(* Logix 5000 project; controller RSL5k_18_Template_noLib Emulate 5570 rev 32.11; software revision 32.02; part 10 of 16 *)
(* tags used below, declared in another part *)
   Inp_UseCVInitVal : ALIAS FOR Wrk_PIDE.CVInitReq;   // 1=Initialize CV to Inp_CVInitValue
   Inp_PVSrcQ : DINT;   // Source and Quality of Inp_PV (enum)
   Inp_PVNotify : DINT;   // PV Alarm Level and Acknowledgement (enum)
   Inp_CVNotify : DINT;   // CV Alarm Level and Acknowledgement (enum)
   Inp_CascSPNotify : DINT;   // Cascade SP Alarm Level and Acknowledgement (enum)
   Inp_IntlkOK : BOOL;   // 1=Interlocks OK, CV can be set
   Inp_NBIntlkOK : BOOL;   // 1=Non-Bypassable Interlocks OK, CV can be set
   Inp_IntlkAvail : BOOL;   // 1 = Interlock Availibility OK
   Cfg_HasRatio : ALIAS FOR Wrk_PIDE.UseRatio;   // 1=Casc Loop Mode is Ratio, 0=Casc Loop Mode is Cascade
   Cfg_InitToMan : ALIAS FOR Wrk_PIDE.ManualAfterInit;   // 1=Go to Manual Loop Mode when an init request is seen
   Cfg_HiHiDevLim : REAL;   // Current High-High Deviation Status Threshold (PVEU)
   Cfg_HiHiDevDB : REAL;   // High-High Devation Status Deadband (PVEU)
   Cfg_HiDevLim : REAL;   // Current High Deviation Status Threshold (PVEU)
   Cfg_HiDevDB : REAL;   // High Devation Status Deadband (PVEU)
   Cfg_LoDevLim : REAL;   // Current Low Deviation Status Threshold (PVEU)
   Cfg_LoDevDB : REAL;   // Low Devation Status Deadband (PVEU)
   Cfg_LoLoDevLim : REAL;   // Current Low-Low Deviation Status Threshold (PVEU)
   Cfg_LoLoDevDB : REAL;   // Low-Low Devation Status Deadband (PVEU)
   Val_PV : REAL;   // Value of Loop PV (PVEU)
   Val_SP : ALIAS FOR Wrk_PIDE.SP;   // Value of SP being used (after ramping and clamping (PVEU)
   SrcQ_IO : DINT;   // Source and Quality of primary I/O (enumeration)
   SrcQ : DINT;   // Source and Quality of primary Val/Sts (enumeration)
   Val_Sts : DINT;   // Loop Status enum: 0=unknown (POoS @ Intlk CV), 1=Manual, 2=Auto, 3=Cascade (no ratio), 4=Ratio
   Val_Fault : DINT;   // Loop Fault: 0=none, 1=PV Uncertain, 22=LoDev, 23=HiDev, 27=LLDev, 28=HHDev, 29=Intlk Trip, 30=SP Fail, 31=PV Fail, 32=CV
   Val_State : DINT;   // Loop State: 0=Man, 1=In DB, 2=Not in DB, 3=SPRamp, 4=CVRamp, 5=Ratio Clamp, 6=SP Clamp, 7=CV Clamp, 8=Windup L, 9=Windup
   Val_NotifyAll : DINT;   // Highest Alarm prio and ack status this object + PV, CV, CascSP (enum)
   Val_UnackAlmC : DINT;   // Count of Unacknowledged Alarms
   Sts_Casc : BOOL;   // 1=Loop Mode is Cascade/Ratio
   Sts_Auto : BOOL;   // 1=Loop Mode is Auto
   Sts_Man : BOOL;   // 1=Loop Mode is Manual
   Sts_Initializing : ALIAS FOR Wrk_PIDE.CVInitializing;   // 1=CV is initializing because of Request from this loop's Secondary
   Sts_WindupHi : ALIAS FOR Wrk_PIDE.WindupHOut;   // 1=This loop winding up High, to Inp_WindupHi of this loop's Primary
   Sts_WindupLo : ALIAS FOR Wrk_PIDE.WindupLOut;   // 1=This loop winding up Low, to Inp_WindupLo of this loop's Primary
   Sts_ZCDBOn : ALIAS FOR Wrk_PIDE.ZCDeadbandOn;   // Deadband Indicator: 1=PV is within ZC deadband and CV will not change
   Sts_RatioClamped : BOOL;   // 1=Selected Ratio (PSet/OSet_Ratio or Inp_OvrdRatio) has been clamped
   Sts_SPBad : ALIAS FOR Wrk_PIDE.SPProgInv;   // 1=SP Value is Bad (quality) or invalid or Casc SP comms fault
   Sts_IntlkSP : BOOL;   // 1=SP Value is being set by shed to Interlock SP
   Sts_SPHeld : BOOL;   // 1=SP Value is being set by shed to hold last good SP
   Sts_SPClamped : BOOL;   // 1=Selected SP is being clamped (for faceplate animation)
   Sts_SPRamping : BOOL;   // 1=SP is ramping toward Val_SPSet, 0=ramp complete
   Sts_PVBad : BOOL;   // 1=PV Value, comms, quality or EU Limitis Bad
   Sts_PVUncertain : BOOL;   // 1=PV Value is Uncertain (quality)
   Sts_FFBad : ALIAS FOR Wrk_PIDE.FFInv;   // 1=Feedforward Term Value is invalid
   Sts_CVBad : BOOL;   // 1=CV Value is Bad (quality) or invalid or CV comms fault
   Sts_HandFdbkBad : ALIAS FOR Wrk_PIDE.HandFBFaulted;   // 1=Hand FB (Tieback) Value is Bad (quality) or invalid or comms fault
   Sts_IntlkCV : BOOL;   // 1=CV Value is being set by shed to Interlock CV
   Sts_CVHeld : BOOL;   // 1=CV Value is being set by shed to hold last good CV
   Sts_CVClamped : BOOL;   // 1=Selected CV is being clamped (for faceplate animation)
   Sts_CVRamping : ALIAS FOR Wrk_PIDE.CVROCAlarm;   // 1=CV is ramping toward Val_CVSet, 0=ramp complete
   Sts_Available : BOOL;   // 1=PID Loop is available for control by automation (Prog)
   Sts_BypActive : BOOL;   // 1=Bypassing Active (Bypassed or Maintenance)
   Sts_NotRdy : BOOL;   // 1=Device Not Ready, see detail bits for reason
   Nrdy_CfgErr : BOOL;   // 1=Device Not Ready: Configuration Error
   Nrdy_Init : BOOL;   // 1=Device Not Ready: Initialized to Manual Mode
   Nrdy_Intlk : BOOL;   // 1=Device Not Ready: Interlock Not OK
   Nrdy_IOFault : BOOL;   // 1=Device Not Ready: I/O Fault (Shed Requires Reset)
   Nrdy_OoS : BOOL;   // 1=Device Not Ready: Out of Service
   Sts_AlmInh : BOOL;   // 1=One or more Alarms Shelved, Disabled or Suppressed
   Sts_Err : BOOL;   // 1=Error in Config: see detail Err bits for reason
   Err_Timer : BOOL;   // 1=Error in Config: Status On-Delay or Off-Delay Time Invalid
   Err_Alarm : BOOL;   // 1=Error in Config: Alarm Severity Invalid
   Err_RatioLim : ALIAS FOR Wrk_PIDE.RatioLimitsInv;   // 1=Error in Config: Ratio Clamping Limits Invalid
   Err_SPLim : ALIAS FOR Wrk_PIDE.SPLimitsInv;   // 1=Error in Config: Setpoint Clamping Limits Invalid
   Err_CVLim : ALIAS FOR Wrk_PIDE.CVLimitsInv;   // 1=Error in Config: CV Clamping Limits Invalid
   Err_PVEU : ALIAS FOR Wrk_PIDE.PVSpanInv;   // 1=Error in Config: PV EU Max/Min Invalid
   Err_CVEU : BOOL;   // 1=Error in Config: CV EU Max/Min Invalid
   Err_CVRaw : ALIAS FOR Wrk_PIDE.CVEUSpanInv;   // 1=Error in Config: CV Raw Max/Min Invalid
   Err_ZCDB : ALIAS FOR Wrk_PIDE.ZCDeadbandInv;   // 1=Error in Config: Loop Zero Crossing Deadband Invalid
   Sts_Hand : ALIAS FOR CmdSrc.Sts_Hand;
   Sts_OoS : ALIAS FOR CmdSrc.Sts_OoS;
   Sts_Prog : ALIAS FOR CmdSrc.Sts_Prog;
   Sts_RdyReset : ALIAS FOR ORdy_Reset;   // 1=A latched alarm or shed condition is ready to be reset
   Sts_RdyAck : BOOL;   // 1=An alarm is ready to be acknowledged
   Sts_HiHiDevCmp : ALIAS FOR HiHiDevGate.Inp;   // High-High Deviation comparison result 1=High-High
   Sts_HiHiDev : ALIAS FOR HiHiDev.Inp;   // 1=PV Deviation is above High-High limit
   Sts_HiDevCmp : ALIAS FOR HiDevGate.Inp;   // High Deviation comparison result 1=High-High
   Sts_HiDev : ALIAS FOR HiDev.Inp;   // 1=PV Deviation is above High limit
   Sts_LoDevCmp : ALIAS FOR LoDevGate.Inp;   // Low Deviation comparison result 1=High-High
   Sts_LoDev : ALIAS FOR LoDev.Inp;   // 1=PV Deviation is below Low limit
   Sts_LoLoDevCmp : ALIAS FOR LoLoDevGate.Inp;   // Low-Low Deviation comparison result 1=High-High
   Sts_LoLoDev : ALIAS FOR LoLoDev.Inp;   // 1=PV Deviation is below Low-Low limit
   Sts_Fail : ALIAS FOR Fail.Inp;   // 1=Loop Failure: PV Bad, SP Bad or CV Comm Failure or Bad
   P_PIDE : BOOL;   // Unique Parameter Name for auto - discovery
   CmdSrc : P_CmdSrc;   // Control / Command Source Selection
   Fail : P_Alarm;   // Loop (SP, PV or CV) Failure Alarm
   IntlkTrip : P_Alarm;   // Interlock Trip Alarm
   Wrk_Notify : DINT;   // Buffer for building Val_Notify
   Wrk_State : DINT;   // Buffer for building Val_State
   Wrk_Sts : DINT;   // Buffer for building Val_Sts
   Wrk_Fault : DINT;   // Buffer for building Val_Fault
   LoLoDev : P_Alarm;   // Low-Low Deviation Alarm
   LoDev : P_Alarm;   // Low Deviation Alarm
   HiDev : P_Alarm;   // High Deviation Alarm
   HiHiDev : P_Alarm;   // High-High Deviation Alarm
   Wrk_IntlkOK : BOOL;   // 1=Interlocks are OK, accounting for bypassing
   Wrk_IntlkTripShed : BOOL;   // Shed Latch for Interlock Not OK
   Wrk_PVFailShed : BOOL;   // Shed Latch for PV Failure
   Wrk_SPFailShed : BOOL;   // Shed Latch for SP Failure
   Wrk_CVFailShed : BOOL;   // Shed Latch for CV Failure
   LoLoDevGate : P_Gate;   // Low-Low Deviation Gate/Delay
   LoDevGate : P_Gate;   // Low Deviation Gate/Delay
   HiDevGate : P_Gate;   // High Deviation Gate/Delay
   HiHiDevGate : P_Gate;   // High-High Deviation Gate/Delay
   Val_Notify : DINT;   // Current Alarm Level and Acknowledgement (enumeration)
   Wrk_SrcQ : DINT;   // Buffer for building Source / Quality enumeration
   Wrk_UnackAlmC : DINT;   // Buffer for building Val_UnackAlmC
   ORdy_ResetAckAll : BOOL;   // 1=At least one Alarm or latched Shed condition requires Reset or Ack
   ORdy_Reset : BOOL;   // 1=Ready for OCmd_Reset (enables HMI button)
   Wrk_PVInfNaN : BOOL;   // 1=PV is infinite or not a number
   Wrk_LoLoDev : BOOL;   // Internal flag: Low-Low Deviation Status
   Wrk_HiHiDev : BOOL;   // Internal flag: High-High Deviation Status
   Wrk_LoDev : BOOL;   // Internal flag: Low Deviation Status
   Wrk_HiDev : BOOL;   // Internal flag: High Deviation Status
   Wrk_Init : BOOL;   // 1=AOI has been initialized
(* P_PIDE, continued *)

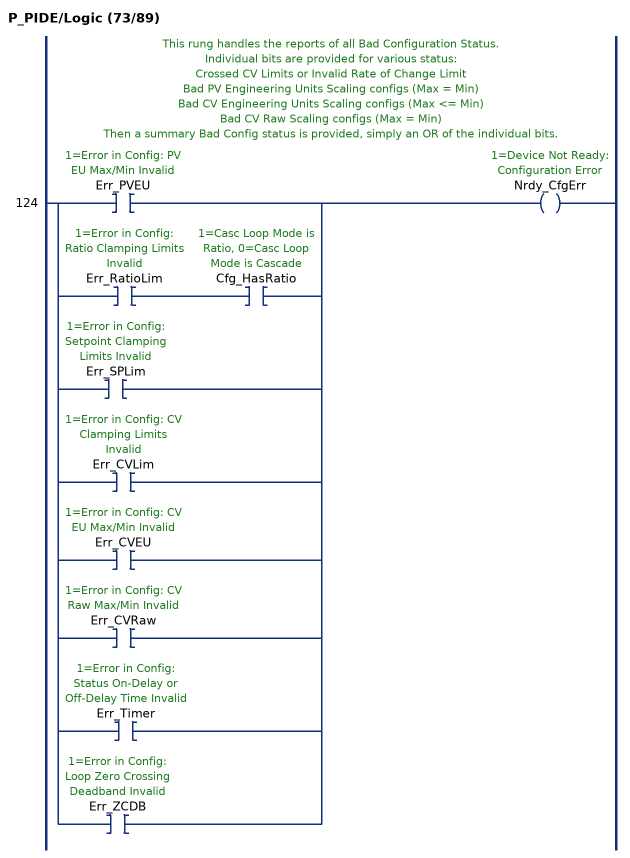
   // This rung handles the reports of all Bad Configuration Status.
   // Individual bits are provided for various status:
   // Crossed CV Limits or Invalid Rate of Change Limit
   // Bad PV Engineering Units Scaling configs (Max = Min)
   // Bad CV Engineering Units Scaling configs (Max <= Min)
   // Bad CV Raw Scaling configs (Max = Min)
   // Then a summary Bad Config status is provided, simply an OR of the individual bits.
   124: [XIC(Err_PVEU) ,XIC(Err_RatioLim) XIC(Cfg_HasRatio) ,XIC(Err_SPLim) ,XIC(Err_CVLim) ,XIC(Err_CVEU) ,XIC(Err_CVRaw) ,XIC(Err_Timer) ,XIC(Err_ZCDB) ]OTE(Nrdy_CfgErr);
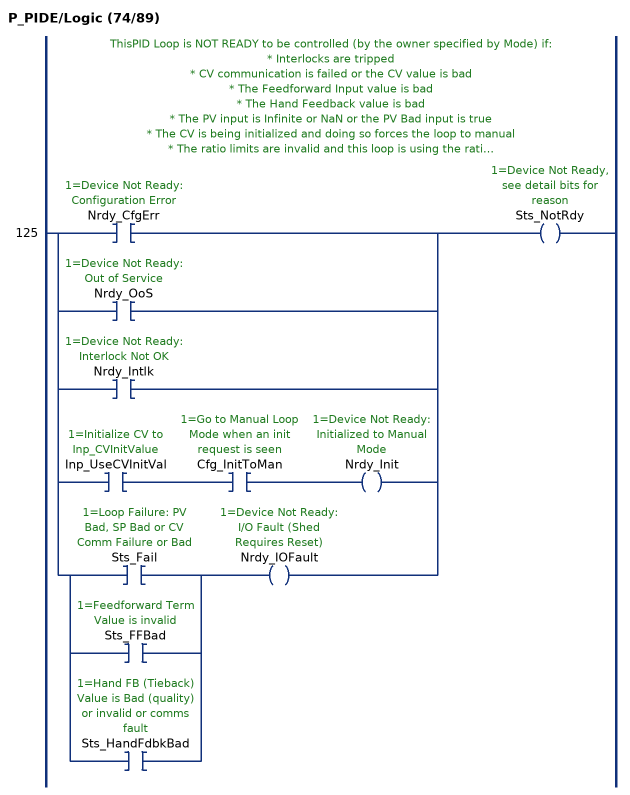
   // ThisPID Loop is NOT READY to be controlled (by the owner specified by Mode) if:
   // * Interlocks are tripped
   // * CV communication is failed or the CV value is bad
   // * The Feedforward Input value is bad
   // * The Hand Feedback value is bad
   // * The PV input is Infinite or NaN or the PV Bad input is true
   // * The CV is being initialized and doing so forces the loop to manual
   // * The ratio limits are invalid and this loop is using the ratio
   // * CV scaling constants are invalid
   // * The instruction is disabled
   // * The setpoint or CV limits are invalid
   // * The instruction is in NO Mode (not owned by anyone)
   125: [XIC(Nrdy_CfgErr) ,XIC(Nrdy_OoS) ,XIC(Nrdy_Intlk) ,XIC(Inp_UseCVInitVal) XIC(Cfg_InitToMan) OTE(Nrdy_Init) ,[XIC(Sts_Fail) ,XIC(Sts_FFBad) ,XIC(Sts_HandFdbkBad) ] OTE(Nrdy_IOFault) ]OTE(Sts_NotRdy);
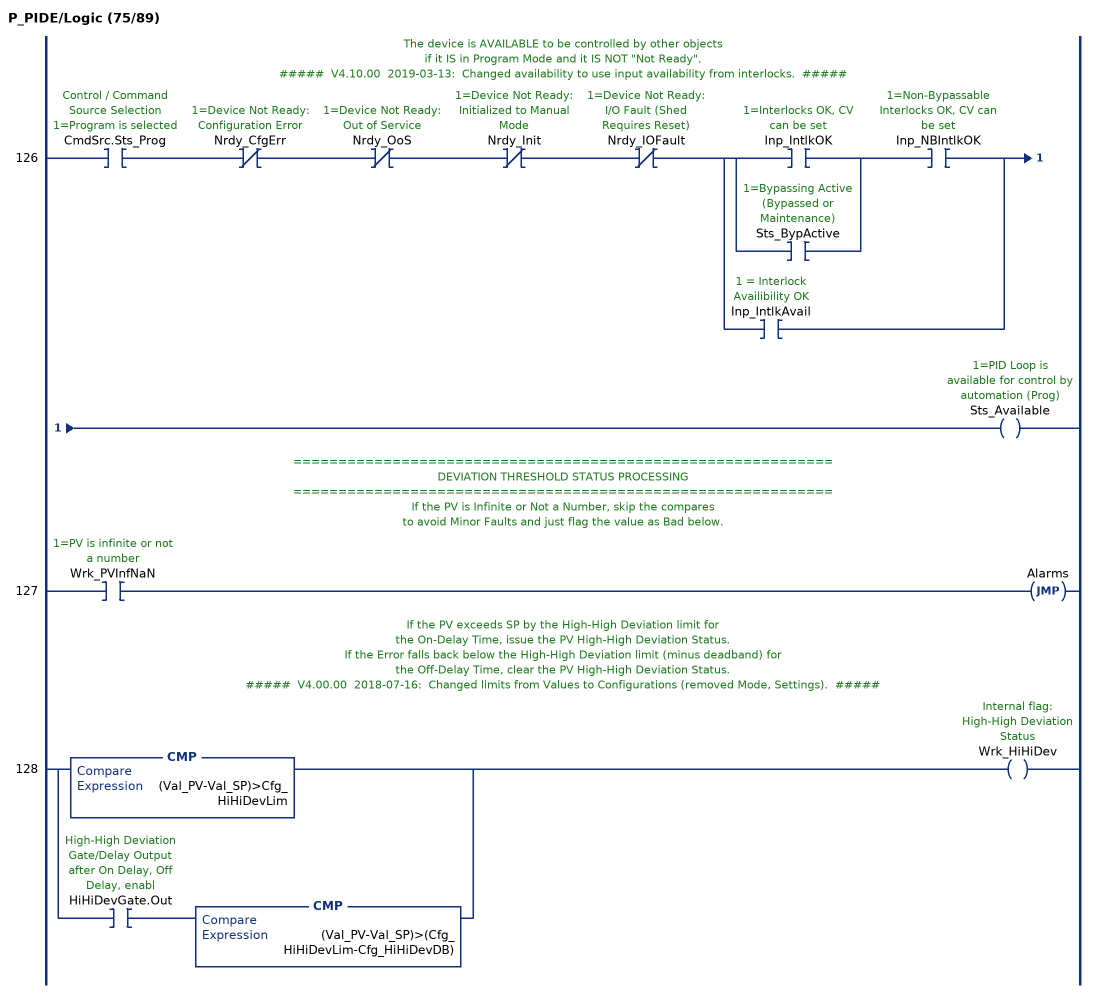
   // The device is AVAILABLE to be controlled by other objects
   // if it IS in Program Mode and it IS NOT "Not Ready".
   // #####  V4.10.00  2019-03-13:  Changed availability to use input availability from interlocks.  #####
   126: XIC(CmdSrc.Sts_Prog)XIO(Nrdy_CfgErr)XIO(Nrdy_OoS)XIO(Nrdy_Init)XIO(Nrdy_IOFault)[[XIC(Inp_IntlkOK) ,XIC(Sts_BypActive) ] XIC(Inp_NBIntlkOK) ,XIC(Inp_IntlkAvail) ]OTE(Sts_Available);
   // ============================================================
   // DEVIATION THRESHOLD STATUS PROCESSING
   // ============================================================
   //  If the PV is Infinite or Not a Number, skip the compares
   // to avoid Minor Faults and just flag the value as Bad below.
   127: XIC(Wrk_PVInfNaN)JMP(Alarms);
   // If the PV exceeds SP by the High-High Deviation limit for
   // the On-Delay Time, issue the PV High-High Deviation Status.
   // If the Error falls back below the High-High Deviation limit (minus deadband) for
   // the Off-Delay Time, clear the PV High-High Deviation Status.
   // #####  V4.00.00  2018-07-16:  Changed limits from Values to Configurations (removed Mode, Settings).  #####
   128: [CMP((Val_PV-Val_SP)>Cfg_HiHiDevLim) ,XIC(HiHiDevGate.Out) CMP((Val_PV-Val_SP)>(Cfg_HiHiDevLim-Cfg_HiHiDevDB)) ]OTE(Wrk_HiHiDev);
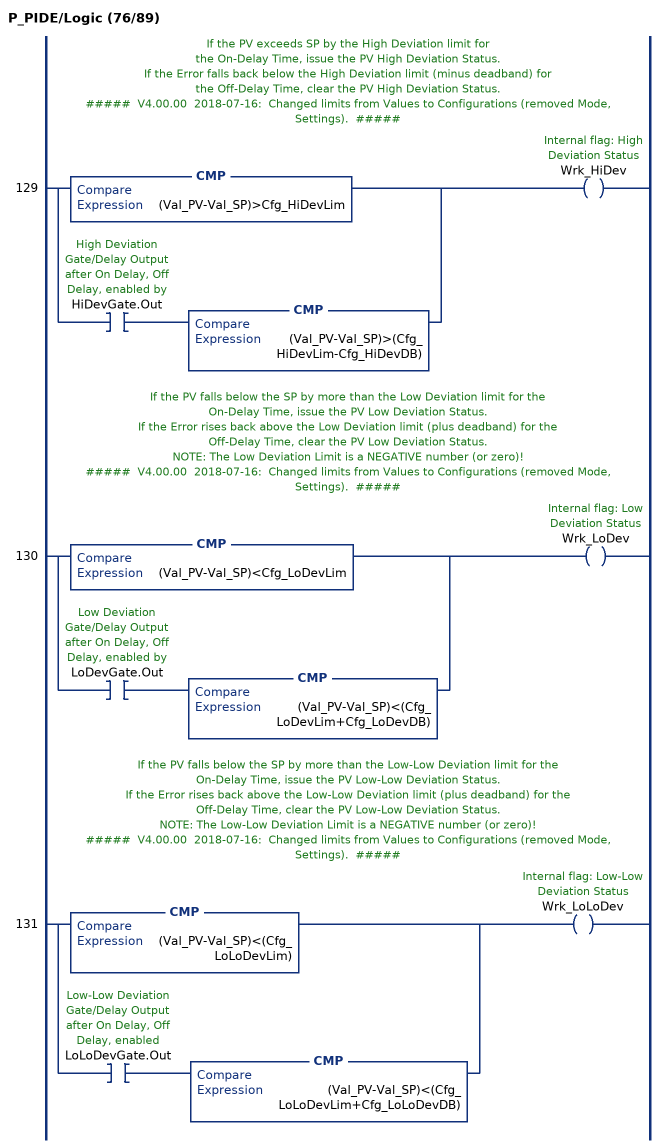
   // If the PV exceeds SP by the High Deviation limit for
   // the On-Delay Time, issue the PV High Deviation Status.
   // If the Error falls back below the High Deviation limit (minus deadband) for
   // the Off-Delay Time, clear the PV High Deviation Status.
   // #####  V4.00.00  2018-07-16:  Changed limits from Values to Configurations (removed Mode, Settings).  #####
   129: [CMP((Val_PV-Val_SP)>Cfg_HiDevLim) ,XIC(HiDevGate.Out) CMP((Val_PV-Val_SP)>(Cfg_HiDevLim-Cfg_HiDevDB)) ]OTE(Wrk_HiDev);
   // If the PV falls below the SP by more than the Low Deviation limit for the
   // On-Delay Time, issue the PV Low Deviation Status.
   // If the Error rises back above the Low Deviation limit (plus deadband) for the
   // Off-Delay Time, clear the PV Low Deviation Status.
   // NOTE: The Low Deviation Limit is a NEGATIVE number (or zero)!
   // #####  V4.00.00  2018-07-16:  Changed limits from Values to Configurations (removed Mode, Settings).  #####
   130: [CMP((Val_PV-Val_SP)<Cfg_LoDevLim) ,XIC(LoDevGate.Out) CMP((Val_PV-Val_SP)<(Cfg_LoDevLim+Cfg_LoDevDB)) ]OTE(Wrk_LoDev);
   // If the PV falls below the SP by more than the Low-Low Deviation limit for the
   // On-Delay Time, issue the PV Low-Low Deviation Status.
   // If the Error rises back above the Low-Low Deviation limit (plus deadband) for the
   // Off-Delay Time, clear the PV Low-Low Deviation Status.
   // NOTE: The Low-Low Deviation Limit is a NEGATIVE number (or zero)!
   // #####  V4.00.00  2018-07-16:  Changed limits from Values to Configurations (removed Mode, Settings).  #####
   131: [CMP((Val_PV-Val_SP)<(Cfg_LoLoDevLim)) ,XIC(LoLoDevGate.Out) CMP((Val_PV-Val_SP)<(Cfg_LoLoDevLim+Cfg_LoLoDevDB)) ]OTE(Wrk_LoLoDev);
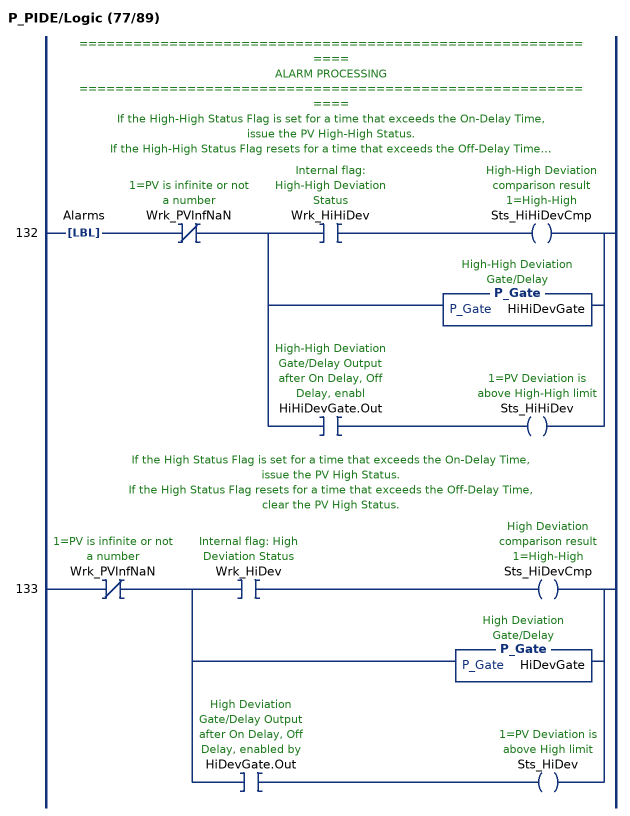
   // ============================================================
   // ALARM PROCESSING
   // ============================================================
   // If the High-High Status Flag is set for a time that exceeds the On-Delay Time,
   // issue the PV High-High Status.
   // If the High-High Status Flag resets for a time that exceeds the Off-Delay Time,
   // clear the PV High-High Status.
   132: LBL(Alarms)XIO(Wrk_PVInfNaN)[XIC(Wrk_HiHiDev) OTE(Sts_HiHiDevCmp) ,P_Gate(HiHiDevGate) ,XIC(HiHiDevGate.Out) OTE(Sts_HiHiDev) ];
   // If the High Status Flag is set for a time that exceeds the On-Delay Time,
   // issue the PV High Status.
   // If the High Status Flag resets for a time that exceeds the Off-Delay Time,
   // clear the PV High Status.
   133: XIO(Wrk_PVInfNaN)[XIC(Wrk_HiDev) OTE(Sts_HiDevCmp) ,P_Gate(HiDevGate) ,XIC(HiDevGate.Out) OTE(Sts_HiDev) ];
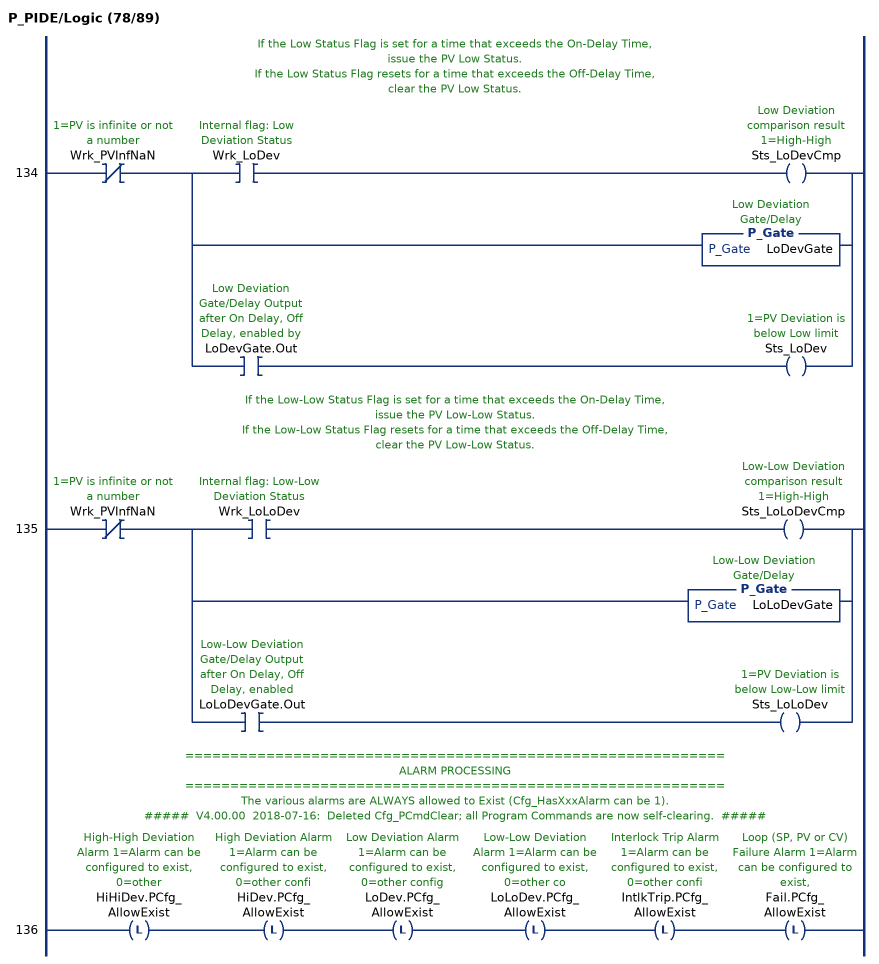
   // If the Low Status Flag is set for a time that exceeds the On-Delay Time,
   // issue the PV Low Status.
   // If the Low Status Flag resets for a time that exceeds the Off-Delay Time,
   // clear the PV Low Status.
   134: XIO(Wrk_PVInfNaN)[XIC(Wrk_LoDev) OTE(Sts_LoDevCmp) ,P_Gate(LoDevGate) ,XIC(LoDevGate.Out) OTE(Sts_LoDev) ];
   // If the Low-Low Status Flag is set for a time that exceeds the On-Delay Time,
   // issue the PV Low-Low Status.
   // If the Low-Low Status Flag resets for a time that exceeds the Off-Delay Time,
   // clear the PV Low-Low Status.
   135: XIO(Wrk_PVInfNaN)[XIC(Wrk_LoLoDev) OTE(Sts_LoLoDevCmp) ,P_Gate(LoLoDevGate) ,XIC(LoLoDevGate.Out) OTE(Sts_LoLoDev) ];
   // ============================================================
   // ALARM PROCESSING
   // ============================================================
   // The various alarms are ALWAYS allowed to Exist (Cfg_HasXxxAlarm can be 1).
   // #####  V4.00.00  2018-07-16:  Deleted Cfg_PCmdClear; all Program Commands are now self-clearing.  #####
   136: OTL(HiHiDev.PCfg_AllowExist)OTL(HiDev.PCfg_AllowExist)OTL(LoDev.PCfg_AllowExist)OTL(LoLoDev.PCfg_AllowExist)OTL(IntlkTrip.PCfg_AllowExist)OTL(Fail.PCfg_AllowExist);
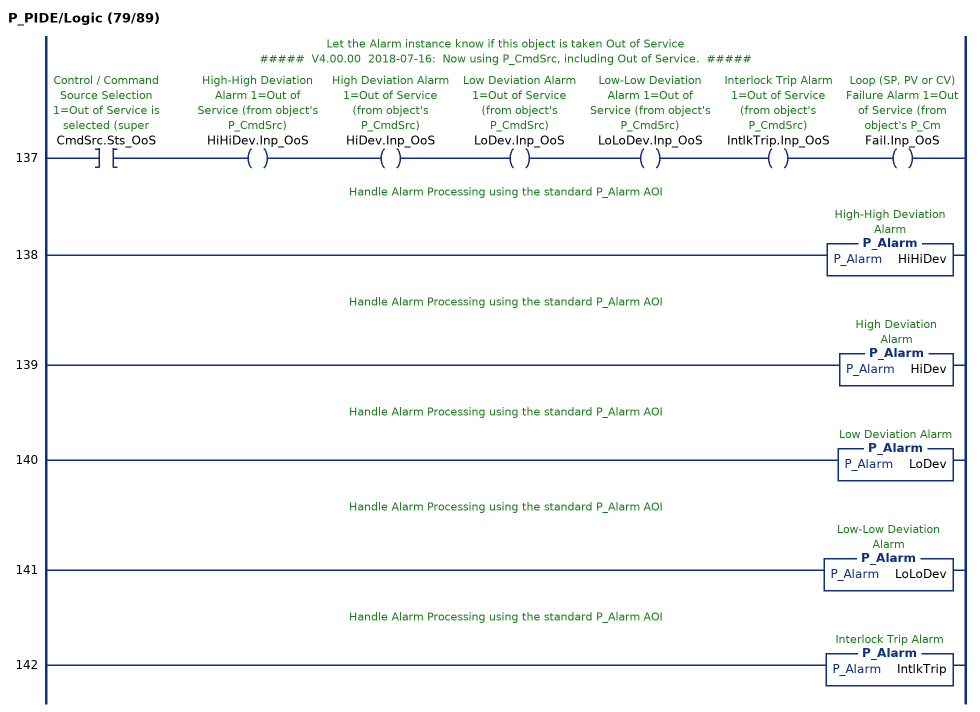
   // Let the Alarm instance know if this object is taken Out of Service
   // #####  V4.00.00  2018-07-16:  Now using P_CmdSrc, including Out of Service.  #####
   137: XIC(CmdSrc.Sts_OoS)OTE(HiHiDev.Inp_OoS)OTE(HiDev.Inp_OoS)OTE(LoDev.Inp_OoS)OTE(LoLoDev.Inp_OoS)OTE(IntlkTrip.Inp_OoS)OTE(Fail.Inp_OoS);
   // Handle Alarm Processing using the standard P_Alarm AOI
   138: P_Alarm(HiHiDev);
   // Handle Alarm Processing using the standard P_Alarm AOI
   139: P_Alarm(HiDev);
   // Handle Alarm Processing using the standard P_Alarm AOI
   140: P_Alarm(LoDev);
   // Handle Alarm Processing using the standard P_Alarm AOI
   141: P_Alarm(LoLoDev);
   // Handle Alarm Processing using the standard P_Alarm AOI
   142: P_Alarm(IntlkTrip);
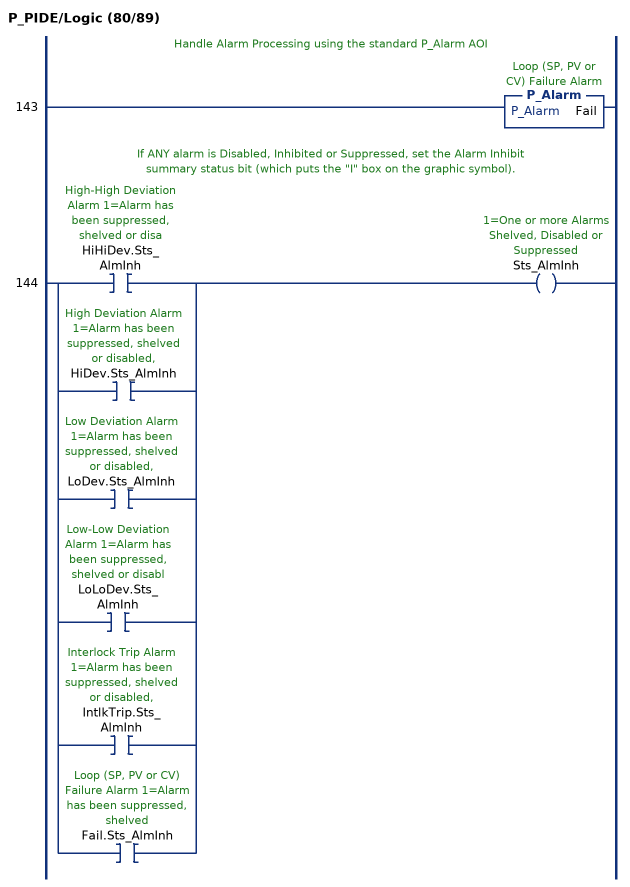
   // Handle Alarm Processing using the standard P_Alarm AOI
   143: P_Alarm(Fail);
   // If ANY alarm is Disabled, Inhibited or Suppressed, set the Alarm Inhibit
   // summary status bit (which puts the "I" box on the graphic symbol).
   144: [XIC(HiHiDev.Sts_AlmInh) ,XIC(HiDev.Sts_AlmInh) ,XIC(LoDev.Sts_AlmInh) ,XIC(LoLoDev.Sts_AlmInh) ,XIC(IntlkTrip.Sts_AlmInh) ,XIC(Fail.Sts_AlmInh) ]OTE(Sts_AlmInh);
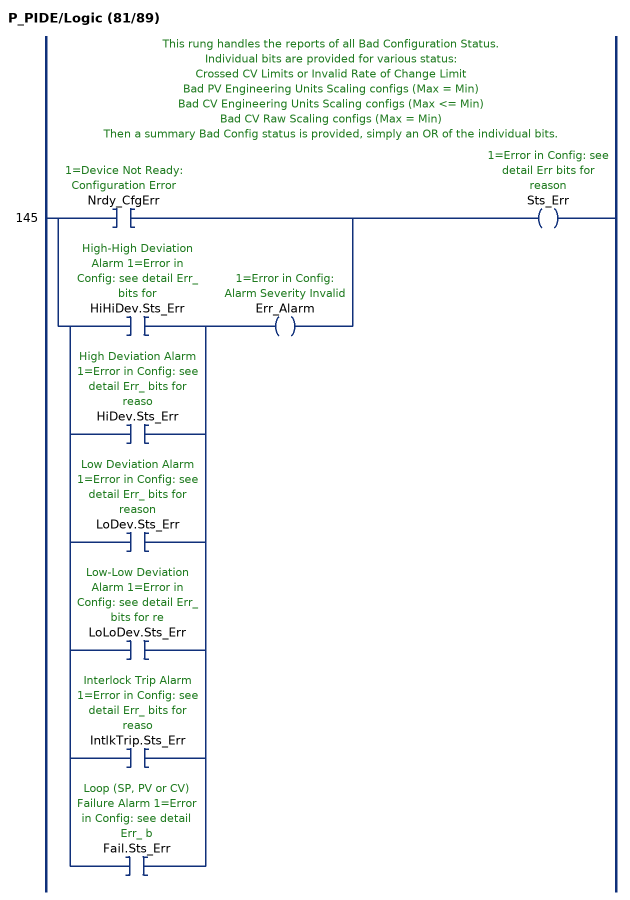
   // This rung handles the reports of all Bad Configuration Status.
   // Individual bits are provided for various status:
   // Crossed CV Limits or Invalid Rate of Change Limit
   // Bad PV Engineering Units Scaling configs (Max = Min)
   // Bad CV Engineering Units Scaling configs (Max <= Min)
   // Bad CV Raw Scaling configs (Max = Min)
   // Then a summary Bad Config status is provided, simply an OR of the individual bits.
   145: [XIC(Nrdy_CfgErr) ,[XIC(HiHiDev.Sts_Err) ,XIC(HiDev.Sts_Err) ,XIC(LoDev.Sts_Err) ,XIC(LoLoDev.Sts_Err) ,XIC(IntlkTrip.Sts_Err) ,XIC(Fail.Sts_Err) ] OTE(Err_Alarm) ]OTE(Sts_Err);
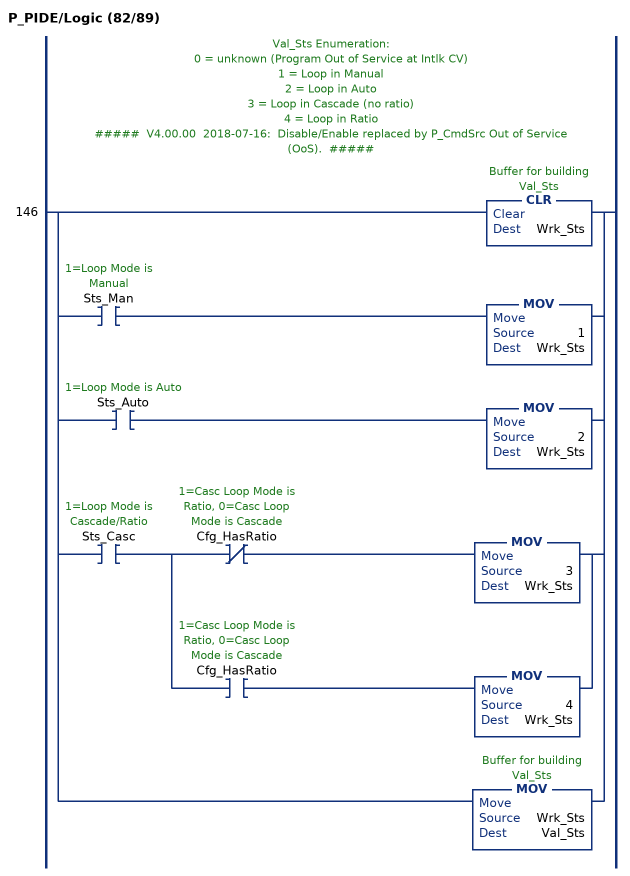
   // Val_Sts Enumeration:
   // 0 = unknown (Program Out of Service at Intlk CV)
   // 1 = Loop in Manual
   // 2 = Loop in Auto
   // 3 = Loop in Cascade (no ratio)
   // 4 = Loop in Ratio
   // #####  V4.00.00  2018-07-16:  Disable/Enable replaced by P_CmdSrc Out of Service (OoS).  #####
   146: [CLR(Wrk_Sts) ,XIC(Sts_Man) MOV(1,Wrk_Sts) ,XIC(Sts_Auto) MOV(2,Wrk_Sts) ,XIC(Sts_Casc) [XIO(Cfg_HasRatio) MOV(3,Wrk_Sts) ,XIC(Cfg_HasRatio) MOV(4,Wrk_Sts) ] ,MOV(Wrk_Sts,Val_Sts) ];
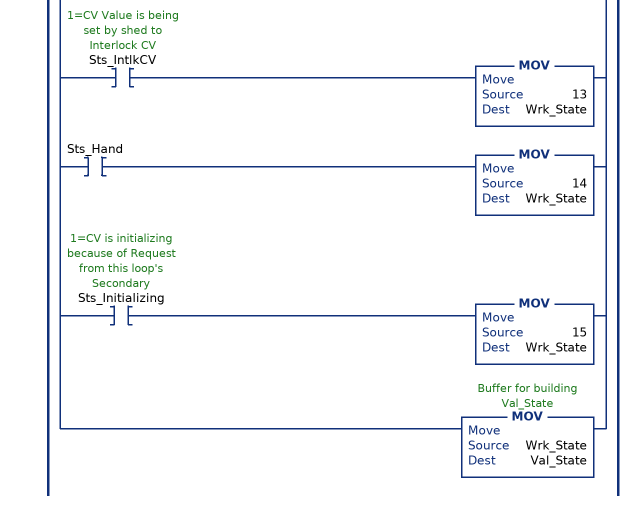
   // Val_State Enumeration:
   // 0 = Manual
   // 1 = Controlled: within deadband
   // 2 = Controlled, not within deadband
   // 3 = Setpoint Ramping
   // 4 = CV Ramping
   // 5 = Ratio Clamped
   // 6 = SP Clamped
   // 7 = CV Clamped
   // 8 = Windup Low
   // 9 = Windup High
   // 10 = SP Held (shed)
   // 11 = SP @ Interlock SP (shed)
   // 12 = CV Held (shed)
   // 13 = CV @ Interlock CV (shed)
   // 14 = CV @ Hand Feedback value
   // 15 = CV Initializing
   147: [CLR(Wrk_State) ,[XIC(Sts_Auto) ,XIC(Sts_Casc) ] [XIC(Sts_ZCDBOn) MOV(1,Wrk_State) ,XIO(Sts_ZCDBOn) MOV(2,Wrk_State) ] ,XIC(Sts_SPRamping) MOV(3,Wrk_State) ,XIC(Sts_CVRamping) MOV(4,Wrk_State) ,XIC(Sts_RatioClamped) MOV(5,Wrk_State) ,XIC(Sts_SPClamped) MOV(6,Wrk_State) ,XIC(Sts_CVClamped) MOV(7,Wrk_State) ,XIC(Sts_WindupLo) MOV(8,Wrk_State) ,XIC(Sts_WindupHi) MOV(9,Wrk_State) ,XIC(Sts_SPHeld) MOV(10,Wrk_State) ,XIC(Sts_IntlkSP) MOV(11,Wrk_State) ,XIC(Sts_CVHeld) MOV(12,Wrk_State) ,XIC(Sts_IntlkCV) MOV(13,Wrk_State) ,XIC(Sts_Hand) MOV(14,Wrk_State) ,XIC(Sts_Initializing) MOV(15,Wrk_State) ,MOV(Wrk_State,Val_State) ];
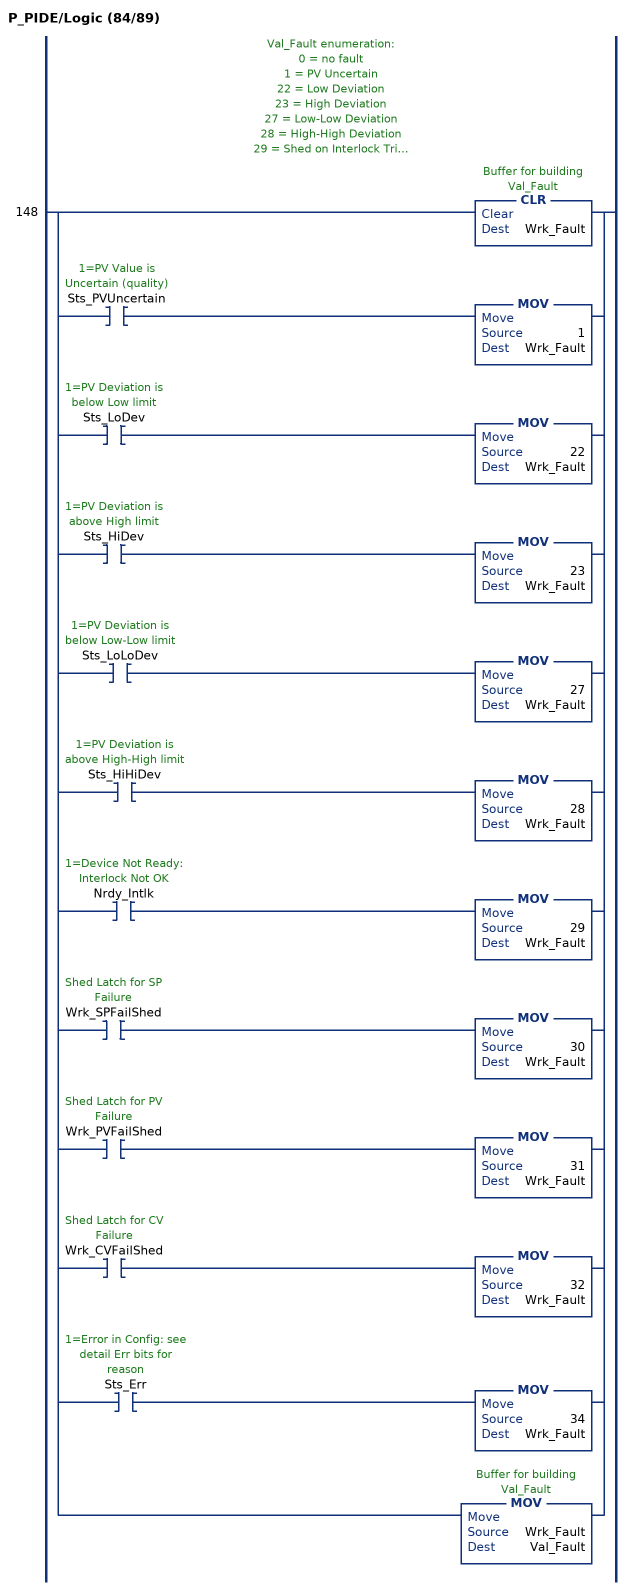
   // Val_Fault enumeration:
   // 0 = no fault
   // 1 = PV Uncertain
   // 22 = Low Deviation
   // 23 = High Deviation
   // 27 = Low-Low Deviation
   // 28 = High-High Deviation
   // 29 = Shed on Interlock Trip
   // 30 = Shed on SP Failure
   // 31 = Shed on PV Failure
   // 32 = Shed on CV Failure
   // 34 = Instruction Configuration Error
   148: [CLR(Wrk_Fault) ,XIC(Sts_PVUncertain) MOV(1,Wrk_Fault) ,XIC(Sts_LoDev) MOV(22,Wrk_Fault) ,XIC(Sts_HiDev) MOV(23,Wrk_Fault) ,XIC(Sts_LoLoDev) MOV(27,Wrk_Fault) ,XIC(Sts_HiHiDev) MOV(28,Wrk_Fault) ,XIC(Nrdy_Intlk) MOV(29,Wrk_Fault) ,XIC(Wrk_SPFailShed) MOV(30,Wrk_Fault) ,XIC(Wrk_PVFailShed) MOV(31,Wrk_Fault) ,XIC(Wrk_CVFailShed) MOV(32,Wrk_Fault) ,XIC(Sts_Err) MOV(34,Wrk_Fault) ,MOV(Wrk_Fault,Val_Fault) ];
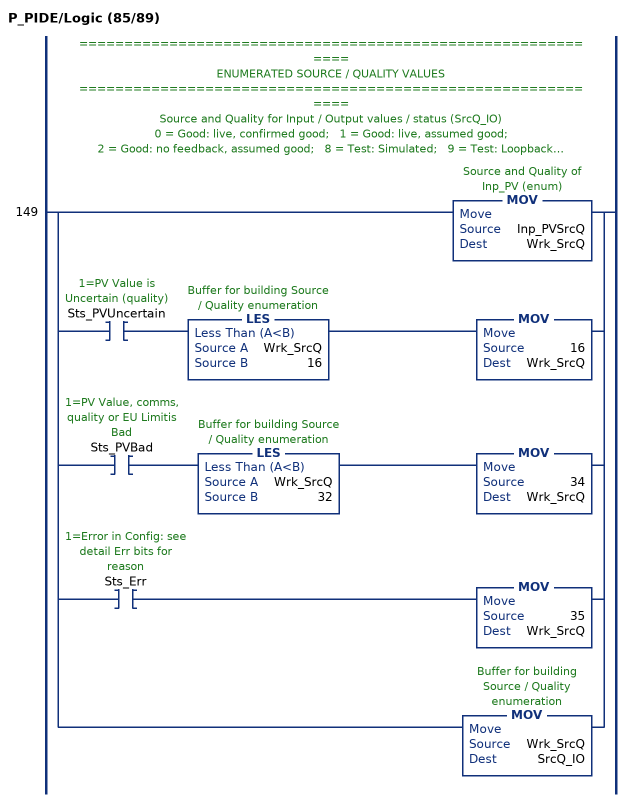
   // ============================================================
   // ENUMERATED SOURCE / QUALITY VALUES
   // ============================================================
   // Source and Quality for Input / Output values / status (SrcQ_IO)
   // 0 = Good: live, confirmed good;   1 = Good: live, assumed good;
   // 2 = Good: no feedback, assumed good;   8 = Test: Simulated;   9 = Test: Loopback;
   // 10 = Test: Manually Entered;   16 = Uncertain: Live, off-spec;
   // 17 = Uncertain, Substituted at Device / Bus;   18 = Uncertain, Substituted at AOI;
   // 19 = Uncertain, using last known good;    20 = Uncertain, using replacement value;
   // 32 = Bad, Signal Failure;   33 = Bad, Channel Fault;
   // 34 = Bad, Module / Comms Fault;   35 = Bad, Invalid Configuration
   149: [MOV(Inp_PVSrcQ,Wrk_SrcQ) ,XIC(Sts_PVUncertain) LES(Wrk_SrcQ,16) MOV(16,Wrk_SrcQ) ,XIC(Sts_PVBad) LES(Wrk_SrcQ,32) MOV(34,Wrk_SrcQ) ,XIC(Sts_Err) MOV(35,Wrk_SrcQ) ,MOV(Wrk_SrcQ,SrcQ_IO) ];
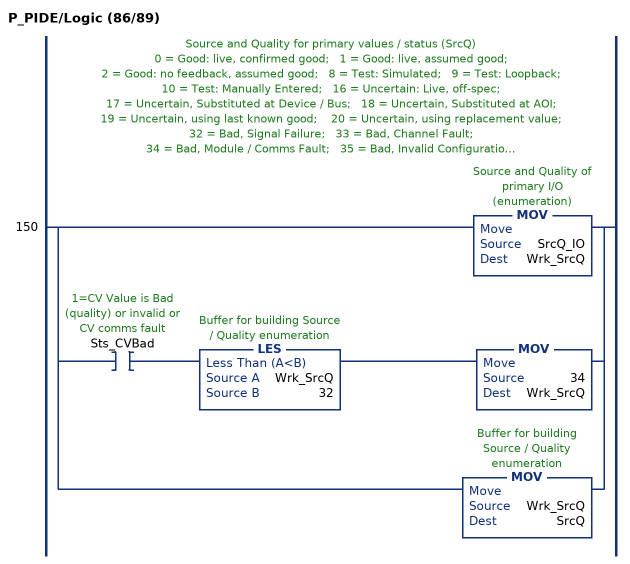
   // Source and Quality for primary values / status (SrcQ)
   // 0 = Good: live, confirmed good;   1 = Good: live, assumed good;
   // 2 = Good: no feedback, assumed good;   8 = Test: Simulated;   9 = Test: Loopback;
   // 10 = Test: Manually Entered;   16 = Uncertain: Live, off-spec;
   // 17 = Uncertain, Substituted at Device / Bus;   18 = Uncertain, Substituted at AOI;
   // 19 = Uncertain, using last known good;    20 = Uncertain, using replacement value;
   // 32 = Bad, Signal Failure;   33 = Bad, Channel Fault;
   // 34 = Bad, Module / Comms Fault;   35 = Bad, Invalid Configuration
   // #####  V4.00.02  2018-12-10:  Modified handling of CV I/O Fault.  #####
   150: [MOV(SrcQ_IO,Wrk_SrcQ) ,XIC(Sts_CVBad) LES(Wrk_SrcQ,32) MOV(34,Wrk_SrcQ) ,MOV(Wrk_SrcQ,SrcQ) ];
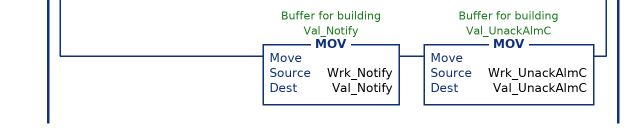
   // ============================================================
   // NOTIFICATION VALUE
   // ============================================================
   // Indicate the current alarm notification level as the max of any of the alarms,
   // and set the low-order bit for reset or ack required:
   // 0 = Not in alarm, acknowledged
   // 1 = Not in alarm, unacknowledged or reset required
   // 2 = Low severity alarm, acknowledged
   // 3 = Low severity alarm, unacknowledged
   // 4 = Medium severity alarm, acknowledged
   // 5 = Medium severity alarm, unacknowledged
   // 6 = High severity alarm, acknowledged
   // 7 = High severity alarm, unacknowledged
   // 8 = Highest severity alarm, acknowledged
   // 9 = Highest severity alarm, unacknowledged
   // #####  V4.00.00  2018-07-16:  Added Val_NotifyAll and Val_UnackAlmC to roll up alarm  #####
   // #####  priority / ack status and unack. alarm count including attached Channel object.  #####
   151: [CLR(Wrk_Notify) CLR(Wrk_UnackAlmC) OTU(Wrk_Notify.0) ,GRT(HiHiDev.Val_Notify,Wrk_Notify) MOV(HiHiDev.Val_Notify,Wrk_Notify) ,GRT(HiDev.Val_Notify,Wrk_Notify) MOV(HiDev.Val_Notify,Wrk_Notify) ,GRT(LoDev.Val_Notify,Wrk_Notify) MOV(LoDev.Val_Notify,Wrk_Notify) ,GRT(LoLoDev.Val_Notify,Wrk_Notify) MOV(LoLoDev.Val_Notify,Wrk_Notify) ,GRT(IntlkTrip.Val_Notify,Wrk_Notify) MOV(IntlkTrip.Val_Notify,Wrk_Notify) ,GRT(Fail.Val_Notify,Wrk_Notify) MOV(Fail.Val_Notify,Wrk_Notify) ,[XIC(HiHiDev.Val_Notify.0) ADD(Wrk_UnackAlmC,1,Wrk_UnackAlmC) ,XIC(HiDev.Val_Notify.0) ADD(Wrk_UnackAlmC,1,Wrk_UnackAlmC) ,XIC(LoDev.Val_Notify.0) ADD(Wrk_UnackAlmC,1,Wrk_UnackAlmC) ,XIC(LoLoDev.Val_Notify.0) ADD(Wrk_UnackAlmC,1,Wrk_UnackAlmC) ,XIC(IntlkTrip.Val_Notify.0) ADD(Wrk_UnackAlmC,1,Wrk_UnackAlmC) ,XIC(Fail.Val_Notify.0) ADD(Wrk_UnackAlmC,1,Wrk_UnackAlmC) ] OTL(Wrk_Notify.0) ,MOV(Wrk_Notify,Val_Notify) MOV(Wrk_UnackAlmC,Val_UnackAlmC) ];
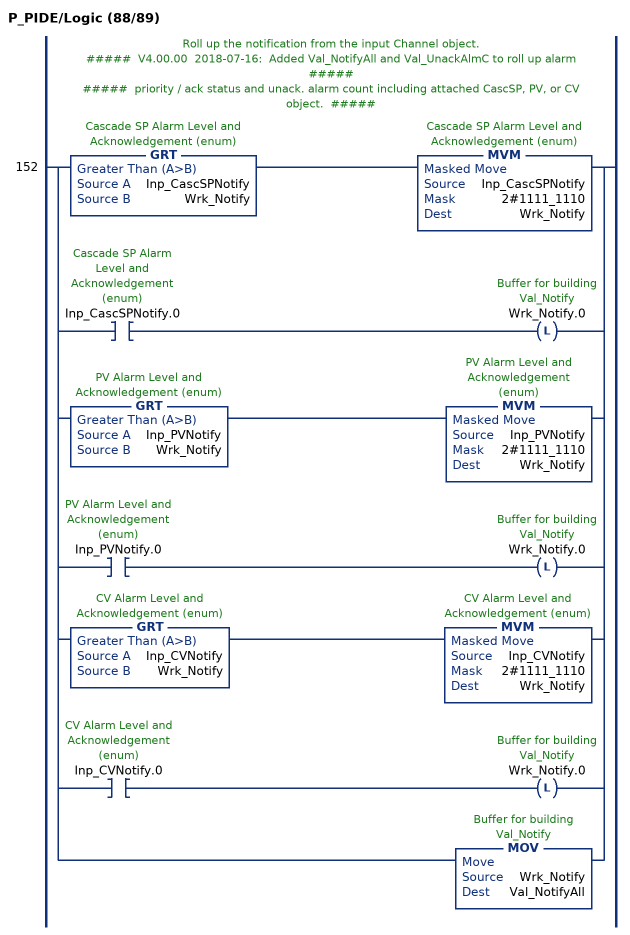
   // Roll up the notification from the input Channel object.
   // #####  V4.00.00  2018-07-16:  Added Val_NotifyAll and Val_UnackAlmC to roll up alarm  #####
   // #####  priority / ack status and unack. alarm count including attached CascSP, PV, or CV object.  #####
   152: [GRT(Inp_CascSPNotify,Wrk_Notify) MVM(Inp_CascSPNotify,2#1111_1110,Wrk_Notify) ,XIC(Inp_CascSPNotify.0) OTL(Wrk_Notify.0) ,GRT(Inp_PVNotify,Wrk_Notify) MVM(Inp_PVNotify,2#1111_1110,Wrk_Notify) ,XIC(Inp_PVNotify.0) OTL(Wrk_Notify.0) ,GRT(Inp_CVNotify,Wrk_Notify) MVM(Inp_CVNotify,2#1111_1110,Wrk_Notify) ,XIC(Inp_CVNotify.0) OTL(Wrk_Notify.0) ,MOV(Wrk_Notify,Val_NotifyAll) ];
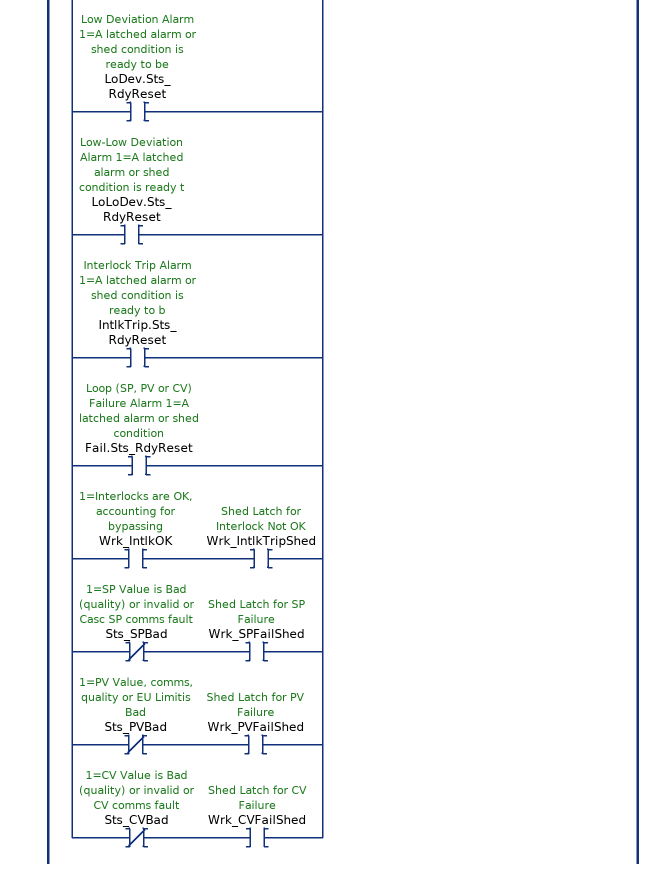
   // This rung identifies:
   // * if a latched Shed condition requires a reset;
   // * if that reset or any alarm reset or other reset is required; and
   // * if any reset or acknowledge from the operator is required.
   // #####  V4.00.00  2018-07-16:  Aligned ready bit naming with command bit names.  #####
   // #####  All OCmds/MCmds and ORdys/MRdys are now Local Tags.  #####
   // #####  Added Sts_RdyAck and Sts_ResetReqd for use by external objects.  #####
   153: [[XIC(HiHiDev.Sts_RdyAck) ,XIC(HiDev.Sts_RdyAck) ,XIC(LoDev.Sts_RdyAck) ,XIC(LoLoDev.Sts_RdyAck) ,XIC(IntlkTrip.Sts_RdyAck) ,XIC(Fail.Sts_RdyAck) ] OTE(Sts_RdyAck) ,[XIC(HiHiDev.Sts_RdyReset) ,XIC(HiDev.Sts_RdyReset) ,XIC(LoDev.Sts_RdyReset) ,XIC(LoLoDev.Sts_RdyReset) ,XIC(IntlkTrip.Sts_RdyReset) ,XIC(Fail.Sts_RdyReset) ,XIC(Wrk_IntlkOK) XIC(Wrk_IntlkTripShed) ,XIO(Sts_SPBad) XIC(Wrk_SPFailShed) ,XIO(Sts_PVBad) XIC(Wrk_PVFailShed) ,XIO(Sts_CVBad) XIC(Wrk_CVFailShed) ] OTE(ORdy_Reset) ]OTE(ORdy_ResetAckAll);
END_ROUTINE

ROUTINE Prescan   (* ladder *)
// Clear Ownership. clear "lurking" Commands, set powerup Loop Mode, SP, and CV per configuration.
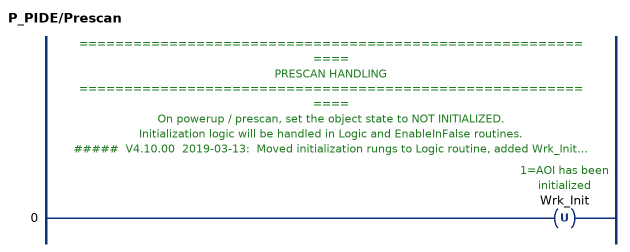
   // ============================================================
   // PRESCAN HANDLING
   // ============================================================
   // On powerup / prescan, set the object state to NOT INITIALIZED.
   // Initialization logic will be handled in Logic and EnableInFalse routines.
   // #####  V4.10.00  2019-03-13:  Moved initialization rungs to Logic routine, added Wrk_Init.  #####
   0: OTU(Wrk_Init);
END_ROUTINE
END_ADD_ON_INSTRUCTION
